FUNCTION_BLOCK SUBSCRIBE_OPCUA_4 (* Composite Function Block Type *)
  (* Standard: 61499-2 *)
  (* Version 1.0, 2019-02-09, iotdeveloperpk *)
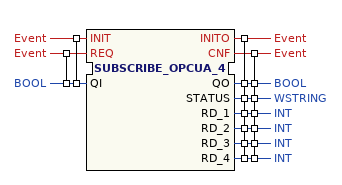
  EVENT_INPUT
    INIT WITH QI; (* Initialization Request *)
    REQ WITH QI; (* Normal Execution Request *)
  END_EVENT
  EVENT_OUTPUT
    INITO WITH QO, STATUS, RD_1, RD_2, RD_3, RD_4; (* Initialization Confirm *)
    CNF WITH QO, STATUS, RD_1, RD_2, RD_3, RD_4; (* Execution Confirmation *)
  END_EVENT
  VAR_INPUT
    QI : BOOL; (* Input event qualifier *)
  END_VAR
  VAR_OUTPUT
    QO : BOOL; (* Output event qualifier *)
    STATUS : WSTRING;
    RD_1 : INT;
    RD_2 : INT;
    RD_3 : INT;
    RD_4 : INT;
  END_VAR
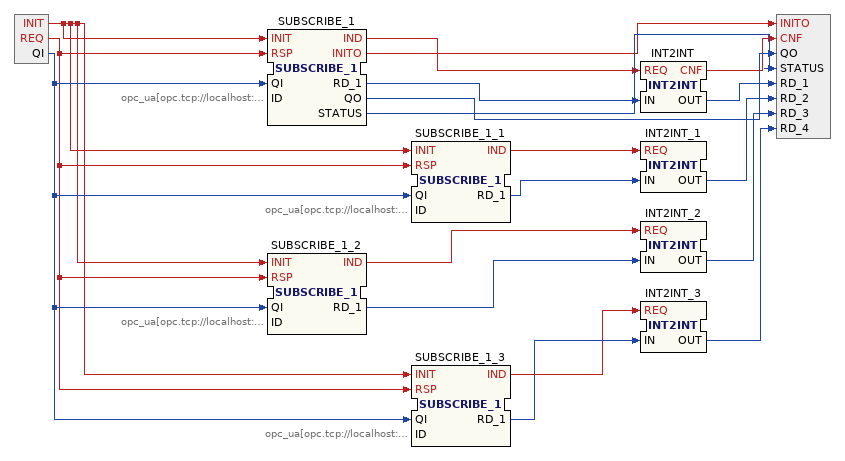
  FBS
    INT2INT : INT2INT;
    INT2INT_1 : INT2INT;
    INT2INT_2 : INT2INT;
    INT2INT_3 : INT2INT;
    SUBSCRIBE_1 : SUBSCRIBE_1(ID := opc_ua[opc.tcp://localhost:4840#/Objects/1:variables/variable1/OUT]);
    SUBSCRIBE_1_1 : SUBSCRIBE_1(ID := opc_ua[opc.tcp://localhost:4840#/Objects/2:variables/variable2/OUT]);
    SUBSCRIBE_1_2 : SUBSCRIBE_1(ID := opc_ua[opc.tcp://localhost:4840#/Objects/3:variables/variable3/OUT]);
    SUBSCRIBE_1_3 : SUBSCRIBE_1(ID := opc_ua[opc.tcp://localhost:4840#/Objects/4:variables/variable4/OUT]);
  END_FBS
  EVENT_CONNECTIONS
    INIT TO SUBSCRIBE_1.INIT;
    INIT TO SUBSCRIBE_1_1.INIT;
    INIT TO SUBSCRIBE_1_2.INIT;
    INIT TO SUBSCRIBE_1_3.INIT;
    REQ TO SUBSCRIBE_1.RSP;
    REQ TO SUBSCRIBE_1_1.RSP;
    REQ TO SUBSCRIBE_1_2.RSP;
    REQ TO SUBSCRIBE_1_3.RSP;
    SUBSCRIBE_1.IND TO INT2INT.REQ;
    SUBSCRIBE_1_1.IND TO INT2INT_1.REQ;
    SUBSCRIBE_1_2.IND TO INT2INT_2.REQ;
    SUBSCRIBE_1_3.IND TO INT2INT_3.REQ;
    SUBSCRIBE_1.INITO TO INITO;
    INT2INT.CNF TO CNF;
  END_CONNECTIONS
  DATA_CONNECTIONS
    SUBSCRIBE_1.RD_1 TO INT2INT.IN;
    SUBSCRIBE_1_1.RD_1 TO INT2INT_1.IN;
    SUBSCRIBE_1_2.RD_1 TO INT2INT_2.IN;
    SUBSCRIBE_1_3.RD_1 TO INT2INT_3.IN;
    QI TO SUBSCRIBE_1.QI;
    QI TO SUBSCRIBE_1_1.QI;
    QI TO SUBSCRIBE_1_2.QI;
    QI TO SUBSCRIBE_1_3.QI;
    SUBSCRIBE_1.QO TO QO;
    SUBSCRIBE_1.STATUS TO STATUS;
    INT2INT.OUT TO RD_1;
    INT2INT_1.OUT TO RD_2;
    INT2INT_2.OUT TO RD_3;
    INT2INT_3.OUT TO RD_4;
  END_CONNECTIONS
END_FUNCTION_BLOCK
